(* PLC project robot6axis, Dassault Systèmes ControlBuild 2024x *)
(* stored: creationDateTime 2023-10-04T11:03:53-01:00 *)

PROGRAM motion_lib.robot6axis
  VAR_INPUT
    armOrigin : ARRAY[1..3] OF REAL := [8705.0, 1630.0, 540.0];
    structRotVectorFOOT : ARRAY[1..3] OF REAL := [0.0, 1.0, 0.0];
    structRotDegFOOT : REAL := -90.01;
    ownRotDegFOOT : REAL := 90.0;
    structRotVectorFOOT2 : ARRAY[1..3] OF REAL := [2(0.0), 1.0];
    structRotDegFOOT2 : REAL := 90.0;
    structRotVectorArm2 : ARRAY[1..3] OF REAL := [2(0.0), 1.0];
    structRotDegArm2 : REAL := -90.0;
    driveRotVector1 : ARRAY[1..3] OF REAL := [1.0, 2(0.0)];
    driveRotVector2 : ARRAY[1..3] OF REAL := [0.0, 1.0, 0.0];
    driveRotVector3 : ARRAY[1..3] OF REAL := [0.0, 1.0, 0.0];
    driveRotVector4 : ARRAY[1..3] OF REAL := [1.0, 2(0.0)];
    driveRotVector5 : ARRAY[1..3] OF REAL := [0.0, 1.0, 0.0];
    driveRotVector6 : ARRAY[1..3] OF REAL := [1.0, 2(0.0)];
    structRotVector1RowA : ARRAY[1..3] OF REAL := [0.0, 1.0, 0.0];
    structRotDeg1RowA : REAL := -90.0;
    structRotVector1RowB : ARRAY[1..3] OF REAL := [0.0, 1.0, 0.0];
    structRotDeg1RowB : REAL := 90.0;
    structRotVectorMultiRowsA : ARRAY[1..3] OF REAL := [0.0, 1.0, 0.0];
    structRotDegMultiRowsA : REAL := 90.0;
    structRotVectorMultiRowsB : ARRAY[1..3] OF REAL := [0.0, 1.0, 0.0];
    structRotDegMultiRowsB : REAL := -90.0;
  END_VAR
  VAR_INPUT
    HomeCmd : BOOL := false;
    MoveVelCmd : BOOL := false;
    MoveAbsCmd : BOOL := false;
    MoveVel1ManualCmd : BOOL := false;
    MoveVel2ManualCmd : BOOL := false;
    MoveAbs1ManualCmd : BOOL := false;
    MoveAbs2ManualCmd : BOOL := false;
    StopCmd : BOOL := false;
    MovePosition : REAL := 0.0;
    MoveSpeed : REAL := 100.0;
    MoveAcceleration : REAL := 100.0;
    MoveDeceleration : REAL := 100.0;
    offsetAxToMa : REAL := 0.0;
  END_VAR
  VAR_INPUT
    HomeCmd2 : BOOL := false;
    MoveVelCmd2 : BOOL := false;
    MoveAbsCmd2 : BOOL := false;
    MoveVel1ManualCmd2 : BOOL := false;
    MoveVel2ManualCmd2 : BOOL := false;
    MoveAbs1ManualCmd2 : BOOL := false;
    MoveAbs2ManualCmd2 : BOOL := false;
    StopCmd2 : BOOL := false;
    MovePosition2 : REAL := 0.0;
    MoveSpeed2 : REAL := 100.0;
    MoveAcceleration2 : REAL := 100.0;
    MoveDeceleration2 : REAL := 100.0;
    offsetAxToMa2 : REAL := 0.0;
  END_VAR
  VAR_INPUT
    HomeCmd3 : BOOL := false;
    MoveVelCmd3 : BOOL := false;
    MoveAbsCmd3 : BOOL := false;
    MoveVel1ManualCmd3 : BOOL := false;
    MoveVel2ManualCmd3 : BOOL := false;
    MoveAbs1ManualCmd3 : BOOL := false;
    MoveAbs2ManualCmd3 : BOOL := false;
    StopCmd3 : BOOL := false;
    MovePosition3 : REAL := 0.0;
    MoveSpeed3 : REAL := 100.0;
    MoveAcceleration3 : REAL := 100.0;
    MoveDeceleration3 : REAL := 100.0;
    offsetAxToMa3 : REAL := 0.0;
  END_VAR
  VAR_INPUT
    HomeCmd4 : BOOL := false;
    MoveVelCmd4 : BOOL := false;
    MoveAbsCmd4 : BOOL := false;
    MoveVel1ManualCmd4 : BOOL := false;
    MoveVel2ManualCmd4 : BOOL := false;
    MoveAbs1ManualCmd4 : BOOL := false;
    MoveAbs2ManualCmd4 : BOOL := false;
    StopCmd4 : BOOL := false;
    MovePosition4 : REAL := 0.0;
    MoveSpeed4 : REAL := 100.0;
    MoveAcceleration4 : REAL := 100.0;
    MoveDeceleration4 : REAL := 100.0;
    offsetAxToMa4 : REAL := 0.0;
  END_VAR
  VAR_INPUT
    HomeCmd5 : BOOL := false;
    MoveVelCmd5 : BOOL := false;
    MoveAbsCmd5 : BOOL := false;
    MoveVel1ManualCmd5 : BOOL := false;
    MoveVel2ManualCmd5 : BOOL := false;
    MoveAbs1ManualCmd5 : BOOL := false;
    MoveAbs2ManualCmd5 : BOOL := false;
    StopCmd5 : BOOL := false;
    MovePosition5 : REAL := 0.0;
    MoveSpeed5 : REAL := 100.0;
    MoveAcceleration5 : REAL := 100.0;
    MoveDeceleration5 : REAL := 100.0;
    offsetAxToMa5 : REAL := 0.0;
  END_VAR
  VAR_INPUT
    HomeCmd6 : BOOL := false;
    MoveVelCmd6 : BOOL := false;
    MoveAbsCmd6 : BOOL := false;
    MoveVel1ManualCmd6 : BOOL := false;
    MoveVel2ManualCmd6 : BOOL := false;
    MoveAbs1ManualCmd6 : BOOL := false;
    MoveAbs2ManualCmd6 : BOOL := false;
    StopCmd6 : BOOL := false;
    MovePosition6 : REAL := 0.0;
    MoveSpeed6 : REAL := 100.0;
    MoveAcceleration6 : REAL := 100.0;
    MoveDeceleration6 : REAL := 100.0;
    offsetAxToMa6 : REAL := 0.0;
  END_VAR
  VAR_INPUT
    PLC_StatusReady : BOOL := true;
    PLC_StatusMoved : BOOL := false;
    PLC_StatusStand : BOOL := false;
    PLC_ActualPositionAx : REAL := 0.0;
    PLC_ActualPositionMa : REAL := 0.0;
    PLC_ActualVelocity : REAL := 0.0;
  END_VAR
  VAR_INPUT
    PLC_StatusReady2 : BOOL := true;
    PLC_StatusMoved2 : BOOL := false;
    PLC_StatusStand2 : BOOL := false;
    PLC_ActualPositionAx2 : REAL := 0.0;
    PLC_ActualPositionMa2 : REAL := 0.0;
    PLC_ActualVelocity2 : REAL := 0.0;
  END_VAR
  VAR_INPUT
    PLC_StatusReady3 : BOOL := true;
    PLC_StatusMoved3 : BOOL := false;
    PLC_StatusStand3 : BOOL := false;
    PLC_ActualPositionAx3 : REAL := 0.0;
    PLC_ActualPositionMa3 : REAL := 0.0;
    PLC_ActualVelocity3 : REAL := 0.0;
  END_VAR
  VAR_INPUT
    PLC_StatusReady4 : BOOL := true;
    PLC_StatusMoved4 : BOOL := false;
    PLC_StatusStand4 : BOOL := false;
    PLC_ActualPositionAx4 : REAL := 0.0;
    PLC_ActualPositionMa4 : REAL := 0.0;
    PLC_ActualVelocity4 : REAL := 0.0;
  END_VAR
  VAR_INPUT
    PLC_StatusReady5 : BOOL := true;
    PLC_StatusMoved5 : BOOL := false;
    PLC_StatusStand5 : BOOL := false;
    PLC_ActualPositionAx5 : REAL := 0.0;
    PLC_ActualPositionMa5 : REAL := 0.0;
    PLC_ActualVelocity5 : REAL := 0.0;
  END_VAR
  VAR_INPUT
    PLC_StatusReady6 : BOOL := true;
    PLC_StatusMoved6 : BOOL := false;
    PLC_StatusStand6 : BOOL := false;
    PLC_ActualPositionAx6 : REAL := 0.0;
    PLC_ActualPositionMa6 : REAL := 0.0;
    PLC_ActualVelocity6 : REAL := 0.0;
  END_VAR
  VAR_INPUT
    gripSyringes : BOOL := false;
  END_VAR
  VAR_OUTPUT
    ActualVelocity1 : REAL := 0.0;
    ActualVelocity2 : REAL := 0.0;
    ActualVelocity3 : REAL := 0.0;
    ActualVelocity4 : REAL := 0.0;
    ActualVelocity5 : REAL := 0.0;
    ActualVelocity6 : REAL := 0.0;
  END_VAR
  VAR_OUTPUT
    armExtrem : ARRAY[1..3] OF REAL := [3(0.0)];
    velX : REAL := 0.0;
    velY : REAL := 0.0;
    velZ : REAL := 0.0;
    armInStop : BOOL := false;
  END_VAR

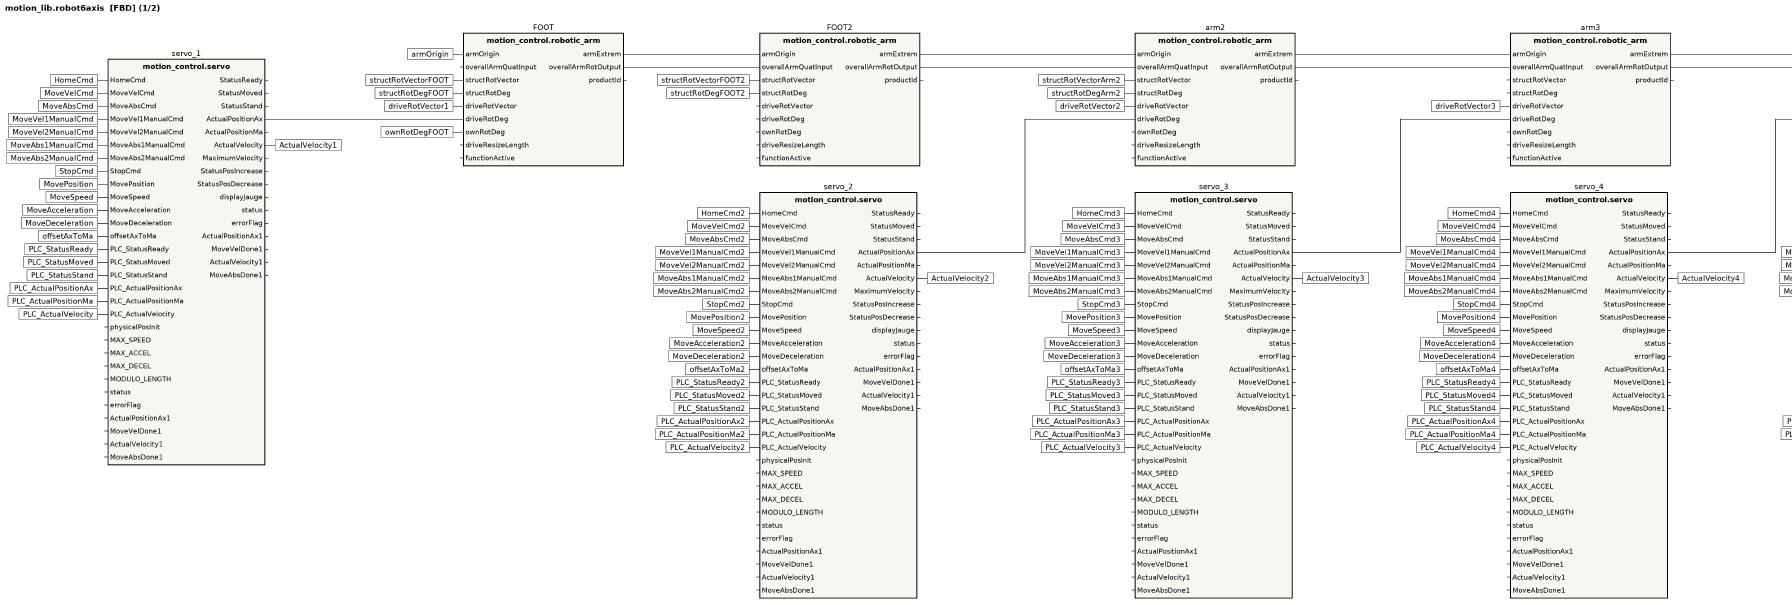
(* FBD diagram, written out as Structured Text *)
servo_1(HomeCmd := HomeCmd, MoveVelCmd := MoveVelCmd, MoveAbsCmd := MoveAbsCmd, MoveVel1ManualCmd := MoveVel1ManualCmd, MoveVel2ManualCmd := MoveVel2ManualCmd, MoveAbs1ManualCmd := MoveAbs1ManualCmd, MoveAbs2ManualCmd := MoveAbs2ManualCmd, StopCmd := StopCmd, MovePosition := MovePosition, MoveSpeed := MoveSpeed, MoveAcceleration := MoveAcceleration, MoveDeceleration := MoveDeceleration, offsetAxToMa := offsetAxToMa, PLC_StatusReady := PLC_StatusReady, PLC_StatusMoved := PLC_StatusMoved, PLC_StatusStand := PLC_StatusStand, PLC_ActualPositionAx := PLC_ActualPositionAx, PLC_ActualPositionMa := PLC_ActualPositionMa, PLC_ActualVelocity := PLC_ActualVelocity);
ActualVelocity1 := servo_1.ActualVelocity;
servo_2(HomeCmd := HomeCmd2, MoveVelCmd := MoveVelCmd2, MoveAbsCmd := MoveAbsCmd2, MoveVel1ManualCmd := MoveVel1ManualCmd2, MoveVel2ManualCmd := MoveVel2ManualCmd2, MoveAbs1ManualCmd := MoveAbs1ManualCmd2, MoveAbs2ManualCmd := MoveAbs2ManualCmd2, StopCmd := StopCmd2, MovePosition := MovePosition2, MoveSpeed := MoveSpeed2, MoveAcceleration := MoveAcceleration2, MoveDeceleration := MoveDeceleration2, offsetAxToMa := offsetAxToMa2, PLC_StatusReady := PLC_StatusReady2, PLC_StatusMoved := PLC_StatusMoved2, PLC_StatusStand := PLC_StatusStand2, PLC_ActualPositionAx := PLC_ActualPositionAx2, PLC_ActualPositionMa := PLC_ActualPositionMa2, PLC_ActualVelocity := PLC_ActualVelocity2);
ActualVelocity2 := servo_2.ActualVelocity;
servo_3(HomeCmd := HomeCmd3, MoveVelCmd := MoveVelCmd3, MoveAbsCmd := MoveAbsCmd3, MoveVel1ManualCmd := MoveVel1ManualCmd3, MoveVel2ManualCmd := MoveVel2ManualCmd3, MoveAbs1ManualCmd := MoveAbs1ManualCmd3, MoveAbs2ManualCmd := MoveAbs2ManualCmd3, StopCmd := StopCmd3, MovePosition := MovePosition3, MoveSpeed := MoveSpeed3, MoveAcceleration := MoveAcceleration3, MoveDeceleration := MoveDeceleration3, offsetAxToMa := offsetAxToMa3, PLC_StatusReady := PLC_StatusReady3, PLC_StatusMoved := PLC_StatusMoved3, PLC_StatusStand := PLC_StatusStand3, PLC_ActualPositionAx := PLC_ActualPositionAx3, PLC_ActualPositionMa := PLC_ActualPositionMa3, PLC_ActualVelocity := PLC_ActualVelocity3);
ActualVelocity3 := servo_3.ActualVelocity;
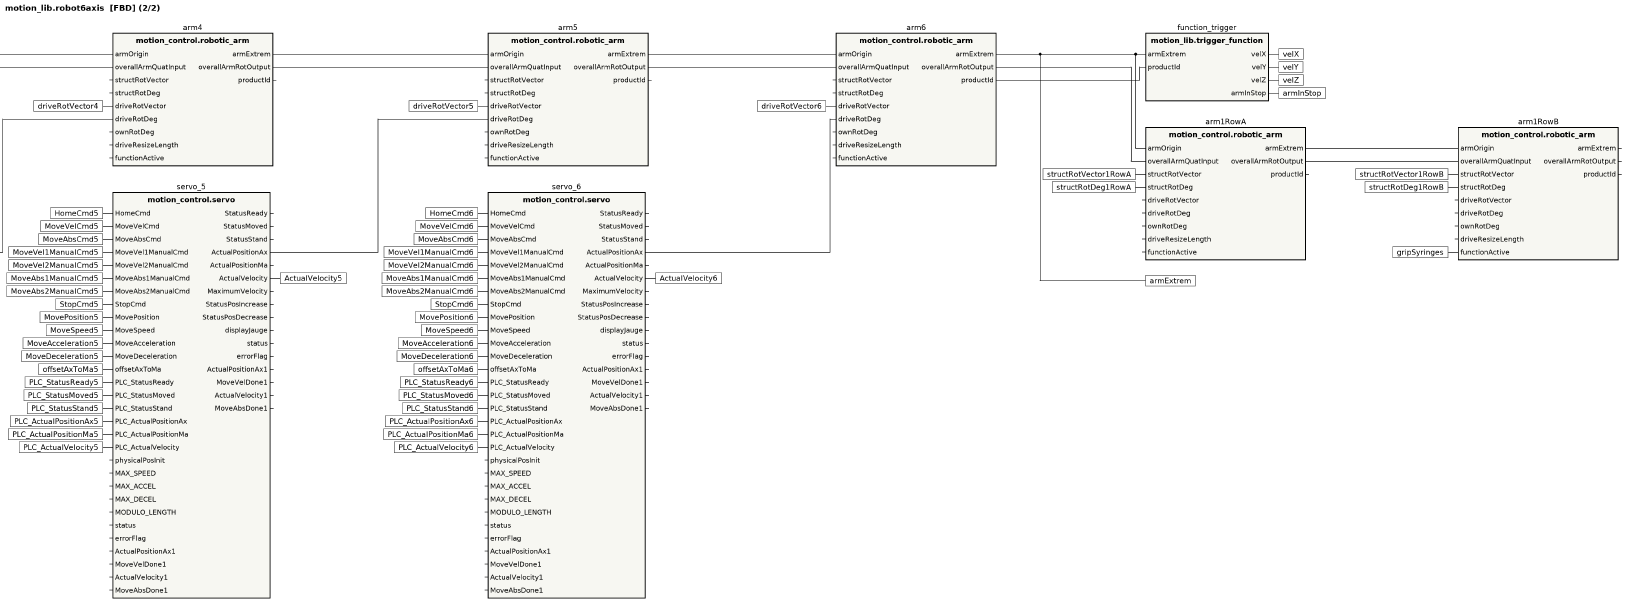
servo_4(HomeCmd := HomeCmd4, MoveVelCmd := MoveVelCmd4, MoveAbsCmd := MoveAbsCmd4, MoveVel1ManualCmd := MoveVel1ManualCmd4, MoveVel2ManualCmd := MoveVel2ManualCmd4, MoveAbs1ManualCmd := MoveAbs1ManualCmd4, MoveAbs2ManualCmd := MoveAbs2ManualCmd4, StopCmd := StopCmd4, MovePosition := MovePosition4, MoveSpeed := MoveSpeed4, MoveAcceleration := MoveAcceleration4, MoveDeceleration := MoveDeceleration4, offsetAxToMa := offsetAxToMa4, PLC_StatusReady := PLC_StatusReady4, PLC_StatusMoved := PLC_StatusMoved4, PLC_StatusStand := PLC_StatusStand4, PLC_ActualPositionAx := PLC_ActualPositionAx4, PLC_ActualPositionMa := PLC_ActualPositionMa4, PLC_ActualVelocity := PLC_ActualVelocity4);
ActualVelocity4 := servo_4.ActualVelocity;
servo_5(HomeCmd := HomeCmd5, MoveVelCmd := MoveVelCmd5, MoveAbsCmd := MoveAbsCmd5, MoveVel1ManualCmd := MoveVel1ManualCmd5, MoveVel2ManualCmd := MoveVel2ManualCmd5, MoveAbs1ManualCmd := MoveAbs1ManualCmd5, MoveAbs2ManualCmd := MoveAbs2ManualCmd5, StopCmd := StopCmd5, MovePosition := MovePosition5, MoveSpeed := MoveSpeed5, MoveAcceleration := MoveAcceleration5, MoveDeceleration := MoveDeceleration5, offsetAxToMa := offsetAxToMa5, PLC_StatusReady := PLC_StatusReady5, PLC_StatusMoved := PLC_StatusMoved5, PLC_StatusStand := PLC_StatusStand5, PLC_ActualPositionAx := PLC_ActualPositionAx5, PLC_ActualPositionMa := PLC_ActualPositionMa5, PLC_ActualVelocity := PLC_ActualVelocity5);
ActualVelocity5 := servo_5.ActualVelocity;
FOOT(armOrigin := armOrigin, structRotVector := structRotVectorFOOT, structRotDeg := structRotDegFOOT, driveRotVector := driveRotVector1, driveRotDeg := servo_1.ActualPositionAx, ownRotDeg := ownRotDegFOOT);
FOOT2(armOrigin := FOOT.armExtrem, overallArmQuatInput := FOOT.overallArmRotOutput, structRotVector := structRotVectorFOOT2, structRotDeg := structRotDegFOOT2);
arm2(armOrigin := FOOT2.armExtrem, overallArmQuatInput := FOOT2.overallArmRotOutput, structRotVector := structRotVectorArm2, structRotDeg := structRotDegArm2, driveRotVector := driveRotVector2, driveRotDeg := servo_2.ActualPositionAx);
arm3(armOrigin := arm2.armExtrem, overallArmQuatInput := arm2.overallArmRotOutput, driveRotVector := driveRotVector3, driveRotDeg := servo_3.ActualPositionAx);
arm4(armOrigin := arm3.armExtrem, overallArmQuatInput := arm3.overallArmRotOutput, driveRotVector := driveRotVector4, driveRotDeg := servo_4.ActualPositionAx);
arm5(armOrigin := arm4.armExtrem, overallArmQuatInput := arm4.overallArmRotOutput, driveRotVector := driveRotVector5, driveRotDeg := servo_5.ActualPositionAx);
servo_6(HomeCmd := HomeCmd6, MoveVelCmd := MoveVelCmd6, MoveAbsCmd := MoveAbsCmd6, MoveVel1ManualCmd := MoveVel1ManualCmd6, MoveVel2ManualCmd := MoveVel2ManualCmd6, MoveAbs1ManualCmd := MoveAbs1ManualCmd6, MoveAbs2ManualCmd := MoveAbs2ManualCmd6, StopCmd := StopCmd6, MovePosition := MovePosition6, MoveSpeed := MoveSpeed6, MoveAcceleration := MoveAcceleration6, MoveDeceleration := MoveDeceleration6, offsetAxToMa := offsetAxToMa6, PLC_StatusReady := PLC_StatusReady6, PLC_StatusMoved := PLC_StatusMoved6, PLC_StatusStand := PLC_StatusStand6, PLC_ActualPositionAx := PLC_ActualPositionAx6, PLC_ActualPositionMa := PLC_ActualPositionMa6, PLC_ActualVelocity := PLC_ActualVelocity6);
arm6(armOrigin := arm5.armExtrem, overallArmQuatInput := arm5.overallArmRotOutput, driveRotVector := driveRotVector6, driveRotDeg := servo_6.ActualPositionAx);
armExtrem := arm6.armExtrem;
ActualVelocity6 := servo_6.ActualVelocity;
function_trigger(armExtrem := arm6.armExtrem, productId := arm6.productId);
velX := function_trigger.velX;
velY := function_trigger.velY;
velZ := function_trigger.velZ;
armInStop := function_trigger.armInStop;
arm1RowA(armOrigin := arm6.armExtrem, overallArmQuatInput := arm6.overallArmRotOutput, structRotVector := structRotVector1RowA, structRotDeg := structRotDeg1RowA);
arm1RowB(armOrigin := arm1RowA.armExtrem, overallArmQuatInput := arm1RowA.overallArmRotOutput, structRotVector := structRotVector1RowB, structRotDeg := structRotDeg1RowB, functionActive := gripSyringes);
END_PROGRAM
